{attribute addProperty BoxType "EL6695-0002-0001"}
{attribute addProperty Id "SYNC_InputsAT %I*SYNC_Inputs_45196B502430IO_InputsEMPTY_STRUCTURE000IO_OutputsEMPTY_STRUCTURE000WcStateAT %I*WcState_98A4DF7520.250InfoDataAT %I*InfoData_275E3363128160"}
{attribute addProperty CRC "2996558720"}
{attribute addProperty SizeInBites "154"}
{attribute addProperty SizeInBytes "19.25"}
TYPE EL6695_5B9A4EC3 :
STRUCT
	{attribute addProperty Name "SYNC_Inputs"}
	SYNC_Inputs : SYNC_Inputs_45196B50;
	{attribute addProperty Name "IO_Inputs"}
	IO_Inputs : EMPTY_STRUCTURE;
	{attribute addProperty Name "IO_Outputs"}
	IO_Outputs : EMPTY_STRUCTURE;
	{attribute addProperty Name "WcState"}
	WcState : WcState_98A4DF75;
	{attribute addProperty Name "InfoData"}
	InfoData : InfoData_275E3363;
END_STRUCT
END_TYPE

(* stored: Version 1.2.0.0, ProductVersion 3.1.4024.9
   DUT EL6695_5B9A4EC3: Id {5c1ed2be-6a3f-41ce-b8bc-d68d70f63cda} *)
